PROGRAM MAIN
VAR

fbReadMB : FB_ReadModbus;
fbMbToVal1: FB_mb_to_val;
fbMbToVal2: FB_mb_to_val;
inputInfo : ARRAY[0..1] OF MODBUS_DATA_MAP :=  [ (_ipAddress := '192.168.1.101', _startAddress:= 0), (_ipAddress := '192.168.1.101', _startAddress:= 12) ];
 
END_VAR


// read and scale XMEAS values to IO
XMEAS_IO[XMEAS_IO_IDX.P_REACTOR]	:= LREAL_TO_INT(32767*(XMEAS[XMEAS_IDX.P_REACTOR]/3000.0));
XMEAS_IO[XMEAS_IO_IDX.L_REACTOR] 	:= LREAL_TO_INT(32767*(XMEAS[XMEAS_IDX.L_REACTOR]/100.0));
//XMEAS_IO[XMEAS_IO_IDX.T_REACTOR] 	:= LREAL_TO_INT(32767*(XMEAS[XMEAS_IDX.T_REACTOR]/175.0));
//XMEAS_IO[XMEAS_IO_IDX.L_SEPARATOR] 	:= LREAL_TO_INT(32767*(XMEAS[XMEAS_IDX.L_SEPARATOR]/100.0));
//XMEAS_IO[XMEAS_IO_IDX.L_STRIPPER] 	:= LREAL_TO_INT(32767*(XMEAS[XMEAS_IDX.L_STRIPPER]/100.0));

//
// BEGIN MODBUS POLLING SEGMENT
//
fbReadMB(inputData := inputInfo );

G_IO.MBS_XMEAS_RAW[1] := fbReadMB.outputData[0];
G_IO.MBS_XMEAS_RAW[2] := fbReadMB.outputData[1];

fbMbToVal1(xi:=G_IO.MBS_XMEAS_RAW[1], i_hi:=20, cal_dc_offset:=G_IO.CAL_XMEAS[1], y_h:=3000.0);
G_IO.MBS_XMEAS[1]:=fbMbToVal1.y;

fbMbToVal2(xi:=G_IO.MBS_XMEAS_RAW[2], i_hi:=20, cal_dc_offset:=G_IO.CAL_XMEAS[2], y_h:=100.0);
G_IO.MBS_XMEAS[2]:=fbMbToVal2.y;

//
// END MODEBUS POLLING SEGMENT
//

END_PROGRAM

(* stored: Version 1.1.0.1, ProductVersion 3.1.0.36
   POU MAIN: Id {a635b5c6-3da2-47b6-922c-5d54bc332cb7}, SpecialFunc None *)
